TYPE stEntity :
STRUCT
	
END_STRUCT
END_TYPE

(* stored: Version 1.1.0.1, ProductVersion 3.1.4024.5
   DUT stEntity: Id {dadae332-a861-4658-9f9b-aa191db89b3e} *)
